PROGRAM MAIN
VAR
	nastro: FB_MSF();
	emg: BOOL;
END_VAR


nastro(
	start:= InputOutput.start, 
	stop:= InputOutput.stop, 
	emg:= InputOutput.emg, 
	ack:= InputOutput.ack, 
	fc1:= InputOutput.fc1, 
	fc2:= InputOutput.fc2, 
	H1=> InputOutput.H1, 
	HEMG=> InputOutput.HEMG, 
	M=> InputOutput.M, 
	libero=> InputOutput.libero);

END_PROGRAM

(* stored: Version 1.1.0.1, ProductVersion 3.1.4024.12
   POU MAIN: Id {026c4556-1d08-4f9d-b723-d4cefff0be76}, SpecialFunc None *)
